{attribute 'qualified_only'}
{attribute 'strict'}
TYPE E_LoadClass :
(
	None:=0,
	Line0,// 优先Line0
	Acquire,// 优先接驳站
	Sensor // 优先传感器检测
);
END_TYPE

(* stored: Version 1.1.0.1, ProductVersion 3.1.4024.3
   DUT E_LoadClass: Id {b747dc3c-61b4-457f-93dd-7a14c840d8ef} *)
